(* IEC 61131-3 sources: matiec-cmake/tests/fixtures, 1 file *)

(* ---- simple_program.st ---- *)
(* Simple test program for fixture testing *)
PROGRAM fixture_test
VAR
    counter : INT := 0;
END_VAR
    counter := counter + 1;
END_PROGRAM
